(* Logix 5000 project; controller pruebaAPM Emulate 5570 rev 30.12; software revision 30.00 *)

TASK MainTask (continuous, watchdog 500 ms) : MainProgram

MODULES
   Local : Emulate 5570 (ICP 2, rev 30.12)
      I_O : vendor 1 type 0 code 15 (ICP 3, rev 1.1, Output RPI 3 ms)
END_MODULES

VAR_GLOBAL   (* controller tags *)
   Banda1 : BOOL;   // Banda de Secado
   Banda2 : BOOL;   // Banda del Enfilador
   Banda3 : BOOL;   // Banda de Seleccion
   BandaPeso : BOOL;
   Cilindro1 : BOOL;   // Cilindro calibre 1
   Cilindro2 : BOOL;   // Cilindro calibre 2
   Cilindro3 : BOOL;   // Cilindro calibre 3
   FullStop : BOOL;   // Parada de emergencia
   KM1 : BOOL;
   L : BOOL;   // Alarma Parada de Emergia
   RST : BOOL;   // Boton de reset
   Secadora : BOOL;
   SP : BOOL;   // sensor porximidad peso
   Speso : DINT;   // Sensor de peso
   SSecado : BOOL;   // Sensor de proximidad
   start : BOOL;
   Step_005 : SFC_STEP := (Status := 16#0020_0000, PauseTimer := 1);
   Stobogan : BOOL;
   stop : BOOL;
   Timer1 : DINT;
END_VAR

PROGRAM MainProgram   (* main routine MainRoutine *)
VAR
   Action_000 : SFC_ACTION := (Status := 16#0020_0000, PauseTimer := 1);
   Action_001 : SFC_ACTION := (Status := 16#0020_0000, PauseTimer := 1);
   Action_002 : SFC_ACTION := (Status := 16#0020_0000, PauseTimer := 1);
   Action_003 : SFC_ACTION := (Status := 16#0020_0000, PauseTimer := 1);
   Action_004 : SFC_ACTION := (Status := 16#0020_0000, PauseTimer := 1);
   Action_005 : SFC_ACTION := (Status := 16#0020_0000, PauseTimer := 1);
   Step_000 : SFC_STEP := (Status := 16#0020_0000, PauseTimer := 1);
   Step_001 : SFC_STEP := (PRE := 3000, TMax := 3050, Count := 2);
   Step_002 : SFC_STEP := (Status := 16#0020_0000, PauseTimer := 1, PRE := 10000, TMax := 10055);
   Step_003 : SFC_STEP := (Status := 16#0020_0000, PauseTimer := 1, T := 8000);
   Step_004 : SFC_STEP := (Status := 16#0020_0000, PauseTimer := 1);
   Step_006 : SFC_STEP := (Status := 16#0020_0000, PauseTimer := 1);
   Step_007 : SFC_STEP := (Status := 16#0020_0000, PauseTimer := 1);
   Step_008 : SFC_STEP := (Status := 16#0020_0000, PauseTimer := 1);
   Step_009 : SFC_STEP := (Status := 16#0020_0000, PauseTimer := 1);
   Tran_000 : BOOL;
   Tran_001 : BOOL;
   Tran_003 : BOOL;
   Tran_004 : BOOL;
   Tran_005 : BOOL;
   Tran_006 : BOOL;
   Tran_007 : BOOL;
END_VAR

ROUTINE MainRoutine   (* ladder *)
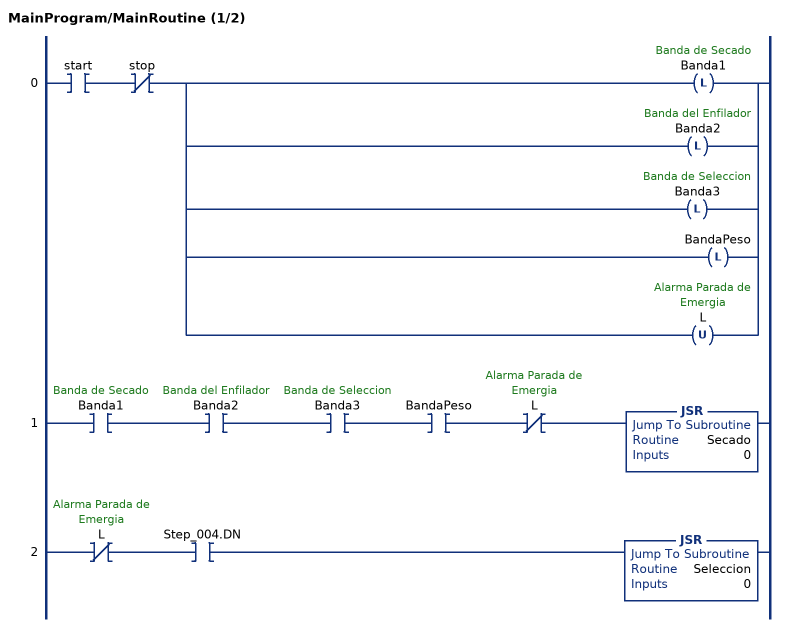
   0: XIC(start)XIO(stop)[OTL(Banda1) ,OTL(Banda2) ,OTL(Banda3) ,OTL(BandaPeso) ,OTU(L) ];
   1: XIC(Banda1)XIC(Banda2)XIC(Banda3)XIC(BandaPeso)XIO(L)JSR(Secado,0);
   2: XIO(L)XIC(Step_004.DN)JSR(Seleccion,0);
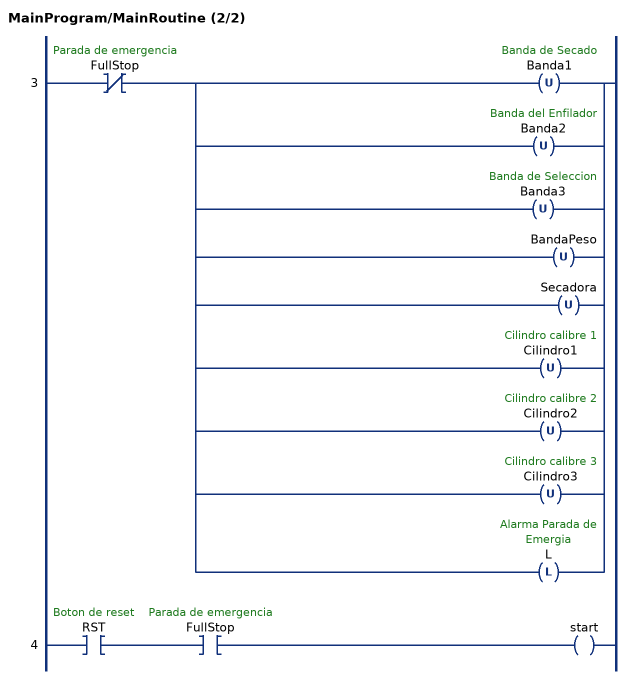
   3: XIO(FullStop)[OTU(Banda1) ,OTU(Banda2) ,OTU(Banda3) ,OTU(BandaPeso) ,OTU(Secadora) ,OTU(Cilindro1) ,OTU(Cilindro2) ,OTU(Cilindro3) ,OTL(L) ];
   4: XIC(RST)XIC(FullStop)OTE(start);
END_ROUTINE

ROUTINE Secado   (* sequential function chart *)
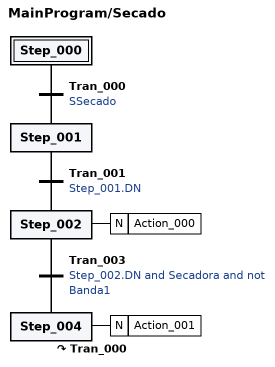
   INITIAL_STEP Step_000:
   END_STEP
   TRANSITION Tran_000 FROM (Step_000, Step_004) TO Step_001
      := SSecado
   END_TRANSITION
   STEP Step_001:
   END_STEP
   TRANSITION Tran_001 FROM Step_001 TO Step_002
      := Step_001.DN
   END_TRANSITION
   STEP Step_002:
      ACTION Action_000 (N):
         Secadora:=1;
         Banda1:=0;
      END_ACTION
   END_STEP
   TRANSITION Tran_003 FROM Step_002 TO Step_004
      := Step_002.DN and Secadora and not Banda1
   END_TRANSITION
   STEP Step_004:
      ACTION Action_001 (N):
         Banda1 := 1;
         Secadora :=0;
      END_ACTION
   END_STEP
END_ROUTINE

ROUTINE Seleccion   (* sequential function chart *)
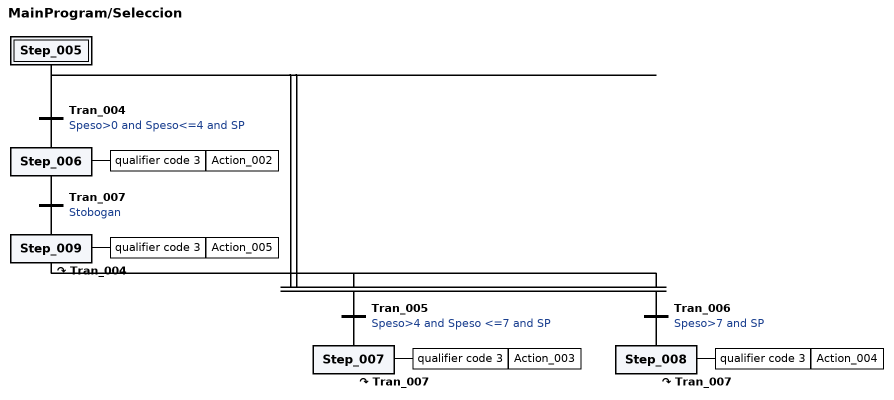
   INITIAL_STEP Step_005:
   END_STEP
   TRANSITION Tran_004 FROM (Step_005, Step_009) TO Step_006
      := Speso>0 and Speso<=4 and SP
   END_TRANSITION
   TRANSITION Tran_005 FROM (Step_005, Step_009) TO Step_007
      := Speso>4 and Speso <=7 and SP
   END_TRANSITION
   TRANSITION Tran_006 FROM (Step_005, Step_009) TO Step_008
      := Speso>7 and SP
   END_TRANSITION
   STEP Step_006:
      ACTION Action_002 (qualifier code 3):
         Cilindro1 :=1;
      END_ACTION
   END_STEP
   STEP Step_007:
      ACTION Action_003 (qualifier code 3):
         Cilindro2 := 1;
      END_ACTION
   END_STEP
   STEP Step_008:
      ACTION Action_004 (qualifier code 3):
         Cilindro3:=1;
      END_ACTION
   END_STEP
   TRANSITION Tran_007 FROM (Step_006, Step_007, Step_008) TO Step_009
      := Stobogan
   END_TRANSITION
   STEP Step_009:
      ACTION Action_005 (qualifier code 3):
         Cilindro1 :=0;
         Cilindro2 :=0;
         Cilindro3 :=0;
      END_ACTION
   END_STEP
END_ROUTINE
END_PROGRAM
